FUNCTION_BLOCK C_BINARYSTREAM IMPLEMENTS I_STREAM
VAR_INPUT
END_VAR
VAR_OUTPUT
END_VAR
VAR
	_MEMBUFFER 	: POINTER TO BYTE;
	_POSITION				: UDINT;
	_PERMISSIBLE_LIMIT 		: UDINT;
	_MEMSIZE	: UDINT;
END_VAR

PROPERTY BufferSize : UDINT
GET
BufferSize := _MEMSIZE;
END_GET
END_PROPERTY

METHOD Close : DINT
VAR_INPUT
END_VAR
IF _MEMBUFFER <> 0 THEN
	__DELETE(_MEMBUFFER);
	_MEMBUFFER := 0;
END_IF
_POSITION := 0;
_PERMISSIBLE_LIMIT := 0;
_MEMSIZE := 0;
END_METHOD

PROPERTY EndOfStream : BOOL
GET
IF _MEMBUFFER <> 0 THEN
	EndOfStream := _POSITION > _PERMISSIBLE_LIMIT;
ELSE
	EndOfStream := TRUE;
END_IF
END_GET
END_PROPERTY

METHOD FB_exit : BOOL
VAR_INPUT
	bInCopyCode : BOOL; // if TRUE, the exit method is called for exiting an instance that is copied afterwards (online change).
END_VAR
IF NOT bInCopyCode THEN
    CLOSE();
END_IF
END_METHOD

PROPERTY IsValid : BOOL
GET
IsValid := _MEMBUFFER <> 0;
END_GET
END_PROPERTY

METHOD New : DINT
VAR_INPUT
	StreamSize	: UDINT;
END_VAR
IF _MEMBUFFER <> 0 THEN
	__DELETE(_MEMBUFFER);
END_IF
_MEMSIZE 				:= StreamSize;
_PERMISSIBLE_LIMIT	 	:= _MEMSIZE - 1;
_POSITION 				:= 0;
_MEMBUFFER 				:= __NEW(BYTE, _MEMSIZE);

New := -1;
RETURN;
END_METHOD

METHOD Peek : DINT
VAR_INPUT
	ptr_DataOut	: POINTER TO BYTE;
END_VAR
IF EndOfStream THEN
	Peek := 1; 
	RETURN;
ELSE
	ptr_DataOut^ := _MEMBUFFER[_POSITION];
	Peek := -1;
	RETURN;
END_IF
END_METHOD

PROPERTY Position : UDINT
GET
POSITION := _POSITION;
END_GET
END_PROPERTY

METHOD Read : DINT
VAR_INPUT
	ptr_DataOut	: PVOID;
	Length		: UDINT;
END_VAR
IF EndOfStream THEN
	Read := 1;
	RETURN;
ELSE
	IF _POSITION + Length > _MEMSIZE THEN
		Read := 1;
		RETURN;
	ELSE
		MEMCPY(ptr_DataOut, _MEMBUFFER + _POSITION, Length);
		_POSITION := _POSITION + Length;
		Read := -1;
		RETURN;
	END_IF
END_IF
END_METHOD

METHOD Seek : DINT
VAR_INPUT
	Offset		: UDINT;	//Permissible range is 0 upto the total buffer size - 1;
	SeekStyle	: E_STREAMSEEKTYPE;
END_VAR
CASE SeekStyle OF 
	//Offsets from the beginning of the stream
	E_STREAMSEEKTYPE.Origin:
		IF Offset > _PERMISSIBLE_LIMIT THEN
			Seek := 1;
			RETURN;
		ELSE
			_POSITION := Offset;
			Seek := -1;
			RETURN;
		END_IF
	//Offsets from the end of the stream
	E_STREAMSEEKTYPE.End:
		IF Offset > _PERMISSIBLE_LIMIT THEN
			Seek := 1;
			RETURN;
		ELSE
			_POSITION := (_PERMISSIBLE_LIMIT) - Offset;
			Seek := -1;
			RETURN;
		END_IF
	//Offsets from the current position of the stream
	E_STREAMSEEKTYPE.Current:
		IF _POSITION + Offset > _PERMISSIBLE_LIMIT THEN
			Seek := 1;
			RETURN;
		ELSE
			_POSITION := _POSITION + Offset;
			Seek := -1;
			RETURN;
		END_IF
END_CASE
END_METHOD

METHOD Write : DINT
VAR_INPUT
	ptr_DataIn	: PVOID;
	Length		: UDINT;
END_VAR
IF EndOfStream THEN
	Write := 1;
	RETURN;
ELSE
	IF _POSITION + Length > _MEMSIZE THEN
		Write := 1;
		RETURN;
	ELSE
		MEMCPY(_MEMBUFFER + _POSITION, ptr_DataIn, Length);
		_POSITION := _POSITION + Length;
		Write := -1;
		RETURN;
	END_IF
END_IF
END_METHOD

END_FUNCTION_BLOCK

(* stored: Version 1.1.0.1, ProductVersion 3.1.4019.2
   POU C_BINARYSTREAM: Id {62e0f9e8-dbe2-4b8a-93c1-515395b38f95}, SpecialFunc None
   Folder Methods: Id {0b2d05ef-671b-442e-8b82-fc2ea9f8c08d}
   Folder internal: Id {54f1fb5c-57f6-41fd-a892-dcc9d93fc6fa}
   Folder Properties: Id {6c6b5bf0-3eda-481e-bfb9-3a069572892e}
   Property BufferSize: Id {e84bbcf7-6c69-4399-a98c-83b895eecd16}
   Get Get: Id {179d321f-648e-4286-8e90-d43f9bcee4db}
   Method Close: Id {08fbbf1f-4aae-4b22-8aa3-912a003574fd}
   Property EndOfStream: Id {6f6204a8-4c51-4744-b888-186b853df35c}
   Get Get: Id {a41f174f-7aeb-44e4-a885-25ef102b07f7}
   Method FB_exit: Id {b11a3324-5538-46dc-8d5f-934cc25c15a1}
   Property IsValid: Id {ccc8adb0-a01a-484e-b272-108dd7287bc0}
   Get Get: Id {b442281c-c63e-4130-a85d-86d73a2f050e}
   Method New: Id {a99da4fd-71fa-4498-bd8a-8613142ce195}
   Method Peek: Id {b55022f1-6b56-4453-a1d2-a9cb27ac413b}
   Property Position: Id {08d8c6ae-ecef-4196-beff-1e8ef3e864f8}
   Get Get: Id {811722b0-cc41-4d04-8f0f-b51038402954}
   Method Read: Id {b4bddcc6-9e3b-4b71-b85e-6d32c4f72b04}
   Method Seek: Id {5dc293f4-09ce-403d-a65e-b36da8ae37a2}
   Method Write: Id {a7b3a4e1-8e6e-49b0-bf17-937a48229722} *)
